Staubli VAL3: onEdit.pgx

public program onEdit(string& x_sItem[] (dimensions=1))
  local string l_sItem
  local string l_sMessage
  local bool l_bContinue
  local string l_sProg
  local num l_nPos
  local num i
  local num l_nSize
  local string l_sPath
  local string l_sButton[2]
begin
  //
  // compose the string
  //
  call language2:getLanguage(l_sPath)
  if l_sPath!=language2:libPath()+"/"+saveData:language
    // set language
    call language2:setLanguage(language2:libPath()+"/"+saveData:language)
  endIf
  //
  l_nPos=find(x_sItem,"PROG")
  call getType(l_sItem)
  if size(x_sItem)>1
    if l_nPos!=-1
      call language2:message(l_sMessage,0)
      l_sProg=right(x_sItem,len(x_sItem)-l_nPos)
      // get the yes_no button Key
      call language:getYesNo(l_sButton)
      // ask the question
      call use:yes_no(l_sItem+" "+x_sItem+"##"+l_sMessage+"#"+l_sProg,l_sButton,l_bContinue)
      if l_bContinue
        x_sItem="Disk://instruction/PROG/page_viewInstr"
        x_sItem[1]=right(l_sProg,len(l_sProg)-len("PROG>"))
      endIf
    else
      popUpMsg(l_sItem+" "+x_sItem)
    endIf
  endIf
end
